TYPE ST_Euchner_MSM_DA_IN :
STRUCT
	///SM_I_X3 | Eingang Zustimmtaster
	bSM_I_X3: BOOL;
	///SM_I_T2 | Eingang Taster
	bSM_I_T2: BOOL;
	///SM_I_T1 | Eingang Taster
	bSM_I_T1: BOOL;
	///SM_E_X3 | Fehler Zustimmtaster
	bSM_E_X3: BOOL;
END_STRUCT
END_TYPE

(* stored: Version 1.1.0.1, ProductVersion 3.1.4024.12
   DUT ST_Euchner_MSM_DA_IN: Id {276d0159-5cd9-4ef0-9cfe-4278d0c90eb0} *)
